ABB RAPID module: Wizard2.modx

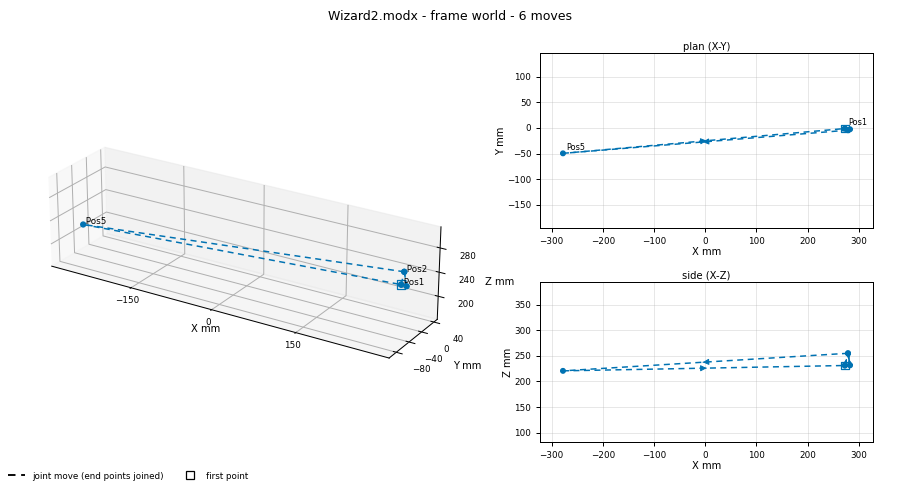
[picture p0: tool path of Wizard2.modx in frame world, 6 of 6 moves have a stored position in this frame; points joined in program order, loops and branches not executed]
MODULE Wizard
PERS robtarget Pos1:=[[272.647705078125, -1.25972330570221, 231.134353637695], [0.344759225845337, 0.536062061786652, -0.767079830169678, -0.07326016575098], [0, -1, -1, 0], [9000000000, 9000000000, 9000000000, 9000000000, 9000000000, 9000000000]];
PERS robtarget Pos2:=[[278.787841796875, -4.46192073822021, 254.970901489258], [0.326371610164642, 0.531330943107605, -0.779361486434937, -0.0613566823303699], [0, -1, -1, 0], [9000000000, 9000000000, 9000000000, 9000000000, 9000000000, 9000000000]];
PERS robtarget Pos3:=[[282.757690429688, -2.70489382743835, 231.48063659668], [0.321605890989304, 0.537844121456146, -0.776510953903198, -0.065757930278778], [0, -1, -1, 0], [9000000000, 9000000000, 9000000000, 9000000000, 9000000000, 9000000000]];
PERS robtarget Pos4:=[[54.3004722595215, 78.4076843261719, 581.065307617188], [0.109736435115337, -0.715388536453247, 0.673441708087921, 0.150510683655739], [0, 0, -1, 4], [9000000000, 9000000000, 9000000000, 9000000000, 9000000000, 9000000000]];
PERS robtarget Pos5:=[[-277.678619384766, -49.6937866210938, 220.693176269531], [0.404614865779877, 0.889612257480621, 0.175065740942955, 0.119284577667713], [2, 0, -1, 0], [9000000000, 9000000000, 9000000000, 9000000000, 9000000000, 9000000000]];
	PROC main()
MoveJ Pos1, v1000, fine, tool0;
MoveJ Pos2, v1000, fine, tool0;
MoveJ Pos3, v1000, fine, tool0;
MoveJ Pos2, v1000, fine, tool0;
MoveJ Pos5, v1000, fine, tool0;

MoveJ Pos1, v1000, fine, tool0;

    ENDPROC
ENDMODULE
